DATA_BLOCK "caiji"
{ S7_Optimized_Access := 'FALSE' }
VERSION : 0.1
NON_RETAIN
"modbus_caiji_new"

BEGIN

END_DATA_BLOCK

